// LS Electric XG5000 project: CTUD
// PLC LSPLC
// module base 0 slot 0: 입출력 모듈:XBC-DR30S (DC 24V 입력 18점, 릴레이 출력 12점)

PROGRAM CTUD (task: 스캔 프로그램)

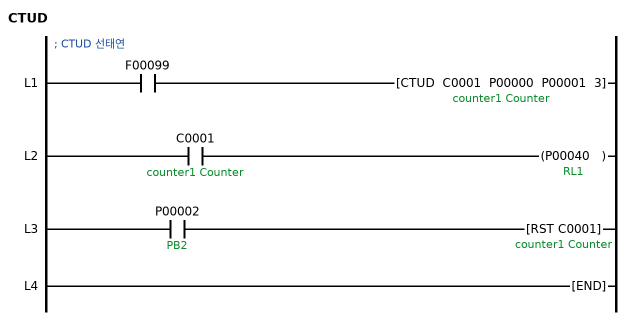
// CTUD 선태연
; L1
LOAD      F00099
CTUD      C0001 P00000 P00001 3	// counter1 Counter
; L2
LOAD      C0001	// counter1 Counter
OUT       P00040	// RL1
; L3
LOAD      P00002	// PB2
RST       C0001	// counter1 Counter
; L4
END